FUNCTION_BLOCK FB_Station
VAR_INPUT
	ifStation:				IF_Station;
	bRstInPos: 				BOOL;
END_VAR
VAR_IN_OUT
	stStationInfo:			ST_Station;
END_VAR
VAR	
	//FBs	
	fbSchrittbetrieb:		FB_Schrittbetrieb;
								
	//Reset
	eResetStatus:			ResetStatus := ResetStatus.bereit;
	bBtnReset:				BOOL;
		
	//Sonstiges
	eInitStatus:			InitStatus := InitStatus.bereit;
	eAblaufStatus:			AblaufStatus := AblaufStatus.bereit;
	
	bTeilBearbeiten:		BOOL;
	nAufnahmeNr:			INT;
	
	bBtnHandZyklus:			BOOL;
END_VAR

//********************************************************************************
//Schrittbetrieb
fbSchrittbetrieb(	eAblaufStatus := eAblaufStatus,
					stStationInfo := stStationInfo,
					bRstInPos := bRstInPos,
					bAblaufAktiv := fbSchrittbetrieb.bAblaufAktiv OR bTeilBearbeiten);
					
fbSchrittbetrieb.bAblaufAktiv := FALSE;

//********************************************************************************					
//Handzyklus
//IF			bBtnHandZyklus THEN
//	bBtnHandZyklus := FALSE;
//	
//	IF			stStationInfo.bZyklusFertig
//		AND		bRstInPos
//		AND NOT MAIN.bProduzieren THEN
//		IF			MAIN.hatAufnBeiStJob(stStationInfo.nStationsNr) THEN							//Aufnahme will bearbeitet werden (Teile wurden schon bestellt)
//			ifStation.bearbeitenAnfordern(MAIN.getAufnahmeBeiStation(stStationInfo.nStationsNr));	//Aktuelle Aufnahme wird verwendet
//		ELSE																						//Aufnahme will NICHT bearbeitet werden (Teile müssen bestellt werden)
//			MAIN.vorwahlPseudoaufnahme();
//			ifStation.bearbeitenAnfordern(Parameter.cAnzAufnahmen+1);								//Pseudoaufnahme wird verwendet
//		END_IF	
//	END_IF
//END_IF

//********************************************************************************					
//Init
IF			stStationInfo.bInit
	AND NOT stStationInfo.bReset THEN
	stStationInfo.bInit := NOT ifStation.init();
END_IF

//********************************************************************************
//Reset
IF			bBtnReset THEN
	bBtnReset := FALSE;
	extReset();
END_IF

IF			stStationInfo.bReset THEN
	stStationInfo.bReset := NOT ifStation.reset();
END_IF

IF		NOT MAIN.bE_NotHalt THEN
	eResetStatus := ResetStatus.bereit;
END_IF

//********************************************************************************					
//Ablauf
IF			stStationInfo.bInitBeendet 
	AND NOT stStationInfo.bReset
	AND NOT fbSchrittbetrieb.bInQueue THEN
	
	IF 			bTeilBearbeiten THEN
		bTeilBearbeiten := NOT ifStation.teilBearbeiten();
	END_IF
END_IF

//********************************************************************************
//Statusanzeige
IF			stStationInfo.bReset THEN
	stStationInfo.sStatus := CONCAT('reset: ', TO_STRING(eResetStatus));
ELSIF			stStationInfo.bInit THEN
	stStationInfo.sStatus := CONCAT('init: ', TO_STRING(eInitStatus));
ELSIF			stStationInfo.bInitBeendet THEN
	stStationInfo.sStatus := TO_STRING(eAblaufStatus);
ELSE
	stStationInfo.sStatus := 'default';
END_IF

METHOD bearbeitenAnfordern
VAR_INPUT
	nAufnahme:		int;
END_VAR
bTeilBearbeiten := TRUE;
nAufnahmeNr := nAufnahme;
END_METHOD

METHOD extReset
VAR_INPUT
END_VAR
eResetStatus := ResetStatus.bereit;			//Reset neu Starten bei jedem Drücken
stStationInfo.bReset := TRUE;
END_METHOD

END_FUNCTION_BLOCK

(* stored: Version 1.1.0.1, ProductVersion 3.1.4026.11
   POU FB_Station: Id {497725e8-26a9-4758-81f0-f8d59e80e301}, SpecialFunc None
   Method bearbeitenAnfordern: Id {bc50bf23-51a4-4fa0-8c91-b17b5b6a500d}
   Method extReset: Id {50aae4f2-5ad8-48b8-9ee5-62fdddd9ddb3} *)
